{attribute 'qualified_only'}
{attribute 'strict'}
{attribute 'to_string'}
TYPE Command :
(
	spleep := 0,
	power,
	move_absolute,
	move_relative,
	move_velocity
)UDINT;
END_TYPE

(* stored: Version 1.1.0.1, ProductVersion 3.1.4026.13
   DUT Command: Id {149475d5-ff6c-4d21-af14-525fed196aaa} *)
